{attribute 'linkalways'} 
{attribute 'no_explicit_call' := 'This FB is a CLASS and must be accessed using methods or properties'}
{attribute 'enable_dynamic_creation'}
FUNCTION_BLOCK _ETcVnRectangleIntersection EXTENDS EnumDatatypeBase
VAR
	localData : ETcVnRectangleIntersection;
	activeData : REFERENCE TO ETcVnRectangleIntersection;
	enumBaseDatatype : _DINT(localData);
END_VAR

METHOD PRIVATE AddLocalEnumeration
VAR_INPUT
	Enumeration : T_MAXSTRING;
	Value : ETcVnRectangleIntersection;
END_VAR
AddEnumeration(Enumeration, Value);
END_METHOD

PROPERTY PUBLIC Address : PVOID
GET
Address := ADR(activeData);
END_GET
END_PROPERTY

METHOD PUBLIC ClearReference
VAR_INPUT
END_VAR
activeData REF= localData;
SetBaseDatatypeReference();
END_METHOD

METHOD PUBLIC Clone : I_Datatype
VAR
    pClone : POINTER TO _ETcVnRectangleIntersection;
END_VAR
pClone := __NEW(_ETcVnRectangleIntersection(InitialValue := Value));
Clone := pClone^;
END_METHOD

METHOD FB_init : BOOL
VAR_INPUT
	bInitRetains : BOOL; // if TRUE, the retain variables are initialized (warm start / cold start)
	bInCopyCode : BOOL;  // if TRUE, the instance afterwards gets moved into the copy code (online change)
	InitialValue : ETcVnRectangleIntersection;
END_VAR
localData := InitialValue;
AddBaseDatatype(enumBaseDatatype);
ClearReference();

AddLocalEnumeration('TCVN_RI_NONE', ETcVnRectangleIntersection.TCVN_RI_NONE);
AddLocalEnumeration('TCVN_RI_PARTIAL', ETcVnRectangleIntersection.TCVN_RI_PARTIAL);
AddLocalEnumeration('TCVN_RI_FULL', ETcVnRectangleIntersection.TCVN_RI_FULL);
END_METHOD

PROPERTY PUBLIC Identifier : T_MAXSTRING
GET
Identifier := 'ETcVnRectangleIntersection';
END_GET
END_PROPERTY

METHOD IsEnumeratorValueEqual : BOOL
VAR_INPUT
	Enumerator : I_KeyValueForwardEnumerator;
END_VAR
VAR
	storedValue : ETcVnRectangleIntersection;
END_VAR
IF NOT Enumerator.TryGet(storedValue) THEN
	RETURN;
END_IF

IsEnumeratorValueEqual := storedValue = activeData;
END_METHOD

METHOD PUBLIC MakeReferenceTo
VAR_INPUT
	ReferenceTarget : REFERENCE TO ETcVnRectangleIntersection;
END_VAR
activeData REF= ReferenceTarget;
SetBaseDatatypeReference();
END_METHOD

METHOD PROTECTED SetBaseDatatypeReference
VAR_INPUT
END_VAR
enumBaseDatatype.MakeReferenceTo(activeData);
END_METHOD

PROPERTY PUBLIC Size : UDINT
GET
Size := SIZEOF(activeData);
END_GET
END_PROPERTY

METHOD TryMakeReferenceTo : BOOL
VAR_INPUT
	Target : I_Datatype;
END_VAR
VAR
	targetAsEnum : I_EnumDatatype;
	pTargetData : POINTER TO ETcVnRectangleIntersection;
END_VAR
IF NOT Target.TryResolveAsEnumDatatype(targetAsEnum) THEN
	RETURN;
END_IF

IF targetAsEnum.Identifier <> Identifier THEN
	RETURN;
END_IF

pTargetData := Target.Address;
activeData REF= pTargetData^;
SetBaseDatatypeReference();
TryMakeReferenceTo := TRUE;
END_METHOD

PROPERTY PUBLIC Value : ETcVnRectangleIntersection
GET
Value := activeData;
END_GET
SET
activeData := Value;
END_SET
END_PROPERTY

END_FUNCTION_BLOCK

(* stored: Version 1.1.0.1, ProductVersion 3.1.4024.12
   POU _ETcVnRectangleIntersection: Id {6c8edae1-72d5-440a-830d-8f4bd01a6f21}, SpecialFunc None
   Folder Constructor: Id {9b27bce5-2caf-4b64-b531-acfb2ba2616d}
   Folder Private: Id {059d35f8-1a64-469f-af8b-4485727ffa1c}
   Folder Protected: Id {3591d3a9-b436-49a5-9b2a-faf58f9c98f7}
   Method AddLocalEnumeration: Id {b091f1ad-60c7-4f5e-9fa2-0ab38ce9cb39}
   Property Address: Id {f44a076a-49e0-4f93-b0f4-2c369cd57e8d}
   Get Get: Id {efd4a1d9-2c12-4996-9aea-bff87b96375f}
   Method ClearReference: Id {b3b8b821-61d9-41f8-8b29-305466bfd283}
   Method Clone: Id {e7a2ce23-9b6a-4aad-8832-bb82b9f4927a}
   Method FB_init: Id {d664bd29-af31-4448-8026-0d8f7ae5e995}
   Property Identifier: Id {fc7112da-665e-469e-8384-a827bdf20edf}
   Get Get: Id {0444fde7-8c26-43e0-b8ec-166cd26e0c91}
   Method IsEnumeratorValueEqual: Id {da3cebca-b9ca-4af3-83cc-3f157e8ac0df}
   Method MakeReferenceTo: Id {f58ca2a4-bb84-45c7-a528-48c6ff675799}
   Method SetBaseDatatypeReference: Id {b294ceab-52a0-46c3-8b94-084b142e77d8}
   Property Size: Id {b411ef27-4887-48d5-ac90-3210c7840e85}
   Get Get: Id {edc3fddd-021a-421f-8e6d-5cdf40fd4a20}
   Method TryMakeReferenceTo: Id {e8377829-62df-4c97-adaf-ce5701092541}
   Property Value: Id {313f008b-b5b2-440b-bee2-83082e98e83b}
   Get Get: Id {e47da6a1-5f7f-4fb7-aa59-8941b43c199d}
   Set Set: Id {a50c8e78-ea30-46f9-8d1c-02dba1d3c73f} *)
